TYPE HmiSlotOccupancy :
STRUCT
	material : STRING;
	occupied : BOOL;
END_STRUCT
END_TYPE

(* stored: Version 1.1.0.1, ProductVersion 3.1.4024.11
   DUT HmiSlotOccupancy: Id {3fe1af31-012a-4c8b-89b1-4b54a3455f56} *)
